FUNCTION_BLOCK FB_TwinSafeConnectionEL3214
(*******************************************************************************************************
Description			:	Evaluate a TwinSAFE connection status and diagnosis to an EtherCAT terminal
Supported terminals : 	EL3214-0090
Documentation 		:	
Version/Date 		:	
Required libraries 	: 	TcSystem.lib (Tc2_System), TcEtherCAT.lib (Tc2_EtherCAT)
********************************************************************************************************)
VAR_INPUT
END_VAR
VAR_OUTPUT

	stInfoData						AT %I*	:ST_TsConnectionInfoEL3214;		(* EL6900 \ Connection Info Data \ Message_X Info Data*)
	nEcSlaveState					AT %I*	:UINT ;							(* EL3214-0090 \ InfoData \ State *)
	stEcAdsAddr						AT %I*	:ST_AdsAddr;					(* EL3214-0090 \ InfoData \ AdsAddr *)

(* act_EcSlaveIdentify *)
	sEcSlaveType							:STRING(15);
	sEcSlaveName							:STRING(31) := '';
	bSlaveIdentify							:BOOL;
	bSlaveTypeError							:BOOL;
	
(* act_Signals *)
	nInSafeDataValue1						:UINT;
	nInSafeDataValue2						:INT;
	nInSafeDataValue3						:INT;
	nInSafeDataValue4						:INT;

(* act_ConnectionState *)
	sState									:STRING;
	
(* act_ConnectionDiag *)
	sDiag									:STRING;
	sFault									:STRING;						(* FailSafe Error (Hardware)*)
	bError									:BOOL;							(* TwinSAFE-Error *)
	
END_VAR
VAR

(* act_ConnectionDiag *)
	nDiag0_3								:BYTE;

(* act_EcSlaveIdentify *)
	fbEcCoeSdoRead							:FB_EcCoESdoReadEx;
	fbEcGetSlaveName						:FB_EcGetSlaveName;

END_VAR
(* End *)

(* Function Block TwinSAFE connection status and diagnosis for EL1904 Terminals *)

(* THIS CODE IS ONLY AN EXAMPLE - YOU HAVE TO CHECK APTITUDE FOR YOUR APPLICATION *)

	(* Identify the EtherCAT slave *)
		act_EcSlaveIdentify();

	(* Evaluate the connection state *)
		act_ConnectionState();
	
	(* Evaluate the connection diagnosis *)
		act_ConnectionDiag();
	
	(* Evaluate the EL3214 input signals *)
		act_Signals();
	
(* End *)

ACTION act_ConnectionDiag:
(* Evaluate the connection diagnosis *)

	(* Evaluate Bit 0..3 *)
	nDiag0_3 := USINT_TO_BYTE(stInfoData.nDiag) AND 16#0F;

	CASE nDiag0_3 OF
		0:		sDiag := 'No error';
		1:		sDiag := 'Invalid command';
		2:		sDiag := 'Unknown command';
		3:		sDiag := 'Invalid connection ID';
		4:		sDiag := 'Invalid CRC';
		5:		sDiag := 'Watchdog time elapsed';
		6:		sDiag := 'Invalid FSOE address';
		7:		sDiag := 'Invalid data';
		8:		sDiag := 'Invalid communication parameter length';
		9:		sDiag := 'Invalid communication parameters';
		10:		sDiag := 'Invalid user parameter length';
		11:		sDiag := 'Invalid user parameter';
		12:		sDiag := 'FSoE master reset';
		13:		sDiag := 'Module err detected on slave, with option "Module error is ComError" activated';
		14:		sDiag := 'Module err detected on EL290x, with option "Error acknowledge active" activated';
		15:		sDiag := 'Slave not yet started, or unexpected error argument';
	END_CASE

	(* Evaluate Bit 4..7 *)
	sFault:='';

	IF stInfoData.nDiag.4 
	THEN
		sFault	:= 'FSoE slave error detected - '; 
	END_IF

	IF stInfoData.nDiag.5 
	THEN
		sFault	:= concat(sFault,'FSoE slave reports Failsafe Value active - ');
	END_IF

	IF stInfoData.nDiag.6 
	THEN
		sFault	:= concat(sFault,'StartUp - ');
	END_IF

	IF stInfoData.nDiag.7 
	THEN
		sFault	:= concat(sFault, 'FSoE master reports Failsafe Value active');
	END_IF
		
	(* Error *)
	bError := stInfoData.nDiag <> 0;

(* End *)
END_ACTION

ACTION act_ConnectionState:
(* Evaluate the connection state *)

	CASE stInfoData.nState OF
		100:	sState := 'Reset state';
		101:	sState := 'Session state';
		102:	sState := 'Connection state';
		103:	sState := 'Parameter state';
		104:	sState := 'Data state';
		105:	sState := 'Shutdown state';
	ELSE
		sState := 'unknown';
	END_CASE
	
(* End *)
END_ACTION

ACTION act_EcSlaveIdentify:
(* Identify the EtherCAT slave *)

	IF NOT nEcSlaveState.3
	THEN
		bSlaveIdentify  := FALSE;
		bSlaveTypeError := FALSE;
		sEcSlaveType    := '';
	END_IF

	IF nEcSlaveState.3
		AND NOT bSlaveIdentify
		AND NOT bSlaveTypeError
 		AND F_CreateAmsNetId(stEcAdsAddr.netId) <> '0.0.0.0.0.0' 
		AND stEcAdsAddr.port <> 0
	THEN

		fbEcCoeSdoRead(
			sNetId			:= 	F_CreateAmsNetId(stEcAdsAddr.netId),
			nSlaveAddr		:= 	stEcAdsAddr.port,
			nSubIndex		:= 	0,
			nIndex			:= 	16#1008,
			pDstBuf			:= 	ADR(sEcSlaveType),
			cbBufLen		:= 	SIZEOF(sEcSlaveType),
			bExecute		:= 	TRUE,
			tTimeout		:= 	DEFAULT_ADS_TIMEOUT);
	

		fbEcGetSlaveName(
			bExecute		:=	TRUE, 
			sNetId			:=	F_CreateAmsNetId(stEcAdsAddr.netId), 
			nSlaveAddr		:=	stEcAdsAddr.port, 
			tTimeout		:=	DEFAULT_ADS_TIMEOUT, 
			bBusy			=>	, 
			sSlaveName		=>	sEcSlaveName, 
			bError			=>	, 
			nErrId			=>	);

		IF NOT fbEcCoeSdoRead.bBusy
			AND NOT fbEcCoeSdoRead.bError
			AND NOT fbEcGetSlaveName.bBusy
			AND NOT fbEcGetSlaveName.bError
		THEN
		
			fbEcCoeSdoRead(bExecute := FALSE); 
			fbEcGetSlaveName(bExecute := FALSE); 

			IF sEcSlaveType = 'EL3214-0090' 
				AND fbEcGetSlaveName.sSlaveName <> ''
			THEN
				bSlaveIdentify := TRUE;
			ELSE
				bSlaveTypeError := TRUE;
			END_IF

		ELSIF NOT fbEcCoeSdoRead.bBusy
			AND fbEcCoeSdoRead.bError
		OR (NOT fbEcGetSlaveName.bBusy
			AND fbEcGetSlaveName.bError)
		THEN
		
			fbEcCoeSdoRead(bExecute := FALSE); 
			fbEcGetSlaveName(bExecute := FALSE); 

		END_IF

	END_IF
	
(* End *)
END_ACTION

ACTION act_Signals:
(* Evaluate the input (EL3214-0090) signals *)

	IF nEcSlaveState.3 (* Slave in operational state *)
	THEN
		(* OP -> transfer the signal states *)
		nInSafeDataValue1 := stInfoData.nInSafeDataValue1;
		nInSafeDataValue2 := stInfoData.nInSafeDataValue2;
		nInSafeDataValue3 := stInfoData.nInSafeDataValue3;
		nInSafeDataValue4 := stInfoData.nInSafeDataValue4;
	ELSE
		(* Error -> clear the signal states *)
		nInSafeDataValue1 := nInSafeDataValue2 := nInSafeDataValue3 := nInSafeDataValue4 := 0;
	END_IF

(* End *)
END_ACTION

END_FUNCTION_BLOCK

(* stored: Version 1.1.0.1, ProductVersion 3.1.4020.12
   POU FB_TwinSafeConnectionEL3214: Id {1434d504-97e3-4f5f-b280-a59effba2168}, SpecialFunc None
   Action act_ConnectionDiag: Id {a3e0ab18-8d4d-4406-b1df-02b8960f7f77}
   Action act_ConnectionState: Id {9cb07e91-0143-4bd5-9ff3-bdcbb34b0008}
   Action act_EcSlaveIdentify: Id {3b1f7f28-ca95-46c1-89ca-a92a7c1efe22}
   Action act_Signals: Id {cc35ef91-734d-465f-b0fa-5cad4b629b80} *)
